FUNCTION F_rad2deg : LREAL
VAR_INPUT
	fInputDeg : LREAL;
END_VAR
VAR
	pi : LREAL := 3.14159265;
END_VAR

F_rad2deg := (180/pi)*fInputDeg;

END_FUNCTION

(* stored: Version 1.1.0.1, ProductVersion 3.1.4024.12
   POU F_rad2deg: Id {3ccf238e-71a2-4e52-88ef-1badeef3e816}, SpecialFunc None *)
